TYPE ST_KinCalcMultiTrafoOut :
STRUCT
    fPos      : ARRAY[1..2] OF ARRAY[1..4] OF LREAL;
    fMetaInfo : ARRAY[1..2] OF U_KinMetaInfo;
END_STRUCT
END_TYPE

(* stored: Version 1.1.0.1
   DUT ST_KinCalcMultiTrafoOut: Id {88b7c0ee-aaa0-4425-bcbe-fe78bc109fb0} *)
